{attribute 'qualified_only'}
VAR_GLOBAL
	bStartButton			: BOOL;
	bStopButton				: BOOL;
END_VAR

(* stored: Version 1.1.0.1, ProductVersion 3.1.4024.11
   GVL IO: Id {a97fe345-8888-4882-81fa-e6a9195840ef} *)
